PROGRAM P_AddrAssignment
VAR
	iDoItOnceCounter	: INT := 0;
END_VAR

CASE iDoItOnceCounter OF
	0: // first cycle after download - assign addresses
		
		GVL_IO.arrStreetLamps[1].eKL6821Module  	:= eKL6821Module_none;
		GVL_IO.arrStreetLamps[1].nAddrShort1		:= 63;
		GVL_IO.arrStreetLamps[1].nAddrShort2		:= 63;
		GVL_IO.arrStreetLamps[1].p_stCommandBuffer	:= ADR(GVL_IO.stCommandBuffer_RB1);
		                                        	
		GVL_IO.arrStreetLamps[2].eKL6821Module  	:= eKL6821Module_RB1;
		GVL_IO.arrStreetLamps[2].nAddrShort1		:= 2;
		GVL_IO.arrStreetLamps[2].nAddrShort2		:= 3;
		GVL_IO.arrStreetLamps[2].p_stCommandBuffer	:= ADR(GVL_IO.stCommandBuffer_RB1);
		                                        	
		GVL_IO.arrStreetLamps[3].eKL6821Module  	:= eKL6821Module_RB1;
		GVL_IO.arrStreetLamps[3].nAddrShort1		:= 0;
		GVL_IO.arrStreetLamps[3].nAddrShort2		:= 1;
		GVL_IO.arrStreetLamps[3].p_stCommandBuffer	:= ADR(GVL_IO.stCommandBuffer_RB1);
		                                        	
		GVL_IO.arrStreetLamps[4].eKL6821Module  	:= eKL6821Module_RB2;
		GVL_IO.arrStreetLamps[4].nAddrShort1		:= 0;
		GVL_IO.arrStreetLamps[4].nAddrShort2		:= 1;
		GVL_IO.arrStreetLamps[4].p_stCommandBuffer	:= ADR(GVL_IO.stCommandBuffer_RB2);
		                                        	
		GVL_IO.arrStreetLamps[5].eKL6821Module  	:= eKL6821Module_RB2;
		GVL_IO.arrStreetLamps[5].nAddrShort1		:= 6;
		GVL_IO.arrStreetLamps[5].nAddrShort2		:= 7;
		GVL_IO.arrStreetLamps[5].p_stCommandBuffer	:= ADR(GVL_IO.stCommandBuffer_RB2);
		                                        	
		GVL_IO.arrStreetLamps[6].eKL6821Module  	:= eKL6821Module_RB2;
		GVL_IO.arrStreetLamps[6].nAddrShort1		:= 3;
		GVL_IO.arrStreetLamps[6].nAddrShort2		:= 5;
		GVL_IO.arrStreetLamps[6].p_stCommandBuffer	:= ADR(GVL_IO.stCommandBuffer_RB2);
		                                        	
		GVL_IO.arrStreetLamps[7].eKL6821Module  	:= eKL6821Module_RB2;
		GVL_IO.arrStreetLamps[7].nAddrShort1		:= 2;
		GVL_IO.arrStreetLamps[7].nAddrShort2		:= 4;
		GVL_IO.arrStreetLamps[7].p_stCommandBuffer	:= ADR(GVL_IO.stCommandBuffer_RB2);
		                                        	
		GVL_IO.arrStreetLamps[8].eKL6821Module  	:= eKL6821Module_RB3;
		GVL_IO.arrStreetLamps[8].nAddrShort1		:= 0;
		GVL_IO.arrStreetLamps[8].nAddrShort2		:= 3;
		GVL_IO.arrStreetLamps[8].p_stCommandBuffer	:= ADR(GVL_IO.stCommandBuffer_RB3);
		                                        	
		GVL_IO.arrStreetLamps[9].eKL6821Module  	:= eKL6821Module_RB3;
		GVL_IO.arrStreetLamps[9].nAddrShort1		:= 1;
		GVL_IO.arrStreetLamps[9].nAddrShort2		:= 2;
		GVL_IO.arrStreetLamps[9].p_stCommandBuffer	:= ADR(GVL_IO.stCommandBuffer_RB3);
		                                        	
		GVL_IO.arrStreetLamps[10].eKL6821Module 	:= eKL6821Module_RB3;
		GVL_IO.arrStreetLamps[10].nAddrShort1		:= 4;
		GVL_IO.arrStreetLamps[10].nAddrShort2		:= 5;
		GVL_IO.arrStreetLamps[10].p_stCommandBuffer	:= ADR(GVL_IO.stCommandBuffer_RB3);
		
		//increment to go to the next step wich is idle
		iDoItOnceCounter := iDoItOnceCounter + 1;
	
	1: // idle state
		; // do nothing
		
END_CASE

END_PROGRAM

(* stored: Version 1.1.0.1, ProductVersion 3.1.4024.5
   POU P_AddrAssignment: Id {dca35f74-e5ff-47a8-a603-2093bdd5e952}, SpecialFunc None *)
